# B&R Automation Studio project TD52 (part 58)

#### MFB50Contr_Lib_private.h
```c
/********************************************************************
 * COPYRIGHT -- Bernecker + Rainer Industrie-Elektronik Ges.m.b.H.
 ********************************************************************
 * Program: MFB50Contr_Lib
 * File: MFB50Contr_Lib_private.h
 * Author: 106001702
 * Created: Wed Nov 09 12:46:00 2011
 ********************************************************************
 * Header for program MFB50Contr_Lib
 ********************************************************************
 * Generated with B&R Automation Studio Target for Simulink V4.2
 * (ERT based)
 ********************************************************************/

#ifndef RTW_HEADER_MFB50Contr_Lib_private_h_
#define RTW_HEADER_MFB50Contr_Lib_private_h_
#include "rtwtypes.h"
#include <bur/plctypes.h>
#ifndef __RTWTYPES_H__
#error This file requires rtwtypes.h to be included
#else
#ifdef TMWTYPES_PREVIOUSLY_INCLUDED
#error This file requires rtwtypes.h to be included before tmwtypes.h
#else

/* Check for inclusion of an incorrect version of rtwtypes.h */
#ifndef RTWTYPES_ID_C08S16I32L32N32F1
#error This code was generated with a different "rtwtypes.h" than the file included
#endif                                 /* RTWTYPES_ID_C08S16I32L32N32F1 */
#endif                                 /* TMWTYPES_PREVIOUSLY_INCLUDED */
#endif                                 /* __RTWTYPES_H__ */

#ifndef MIN
#define MIN(a,b)                       ((a) < (b) ? (a) : (b))
#endif

#ifndef MAX
#define MAX(a,b)                       ((a) > (b) ? (a) : (b))
#endif

/* Imported (extern) block parameters */
extern real_T I0AllCyl[21];            /* Variable: I0AllCyl
                                        * Referenced by: '<Root>/inputvariable'
                                        */
extern real_T MFB50ActAllCyl[21];      /* Variable: MFB50ActAllCyl
                                        * Referenced by: '<Root>/inputvariable8'
                                        */
extern real_T MFB50EnPowTh;            /* Variable: MFB50EnPowTh
                                        * Referenced by: '<Root>/Relay'
                                        */
extern real_T MFB50EnSpdTh;            /* Variable: MFB50EnSpdTh
                                        * Referenced by: '<Root>/default 500 (rpm)'
                                        */
extern real_T MFB50GlobRefExt;         /* Variable: MFB50GlobRefExt
                                        * Referenced by: '<Root>/MFB50RefGlobExt (CADafTDC)'
                                        */
extern real_T MFB50RefOffsetAllCyl[21];/* Variable: MFB50RefOffsetAllCyl
                                        * Referenced by: '<Root>/inputvariable20'
                                        */
extern real_T MapIoP2sx[2];            /* Variable: MapIoP2sx
                                        * Referenced by: '<S7>/inputvariable1'
                                        */
extern real_T MapIoP2sy[2];            /* Variable: MapIoP2sy
                                        * Referenced by: '<S7>/inputvariable2'
                                        */
extern real_T MapMFB50oP2sx[2];        /* Variable: MapMFB50oP2sx
                                        * Referenced by: '<S4>/inputvariable1'
                                        */
extern real_T MapMFB50oP2sy[2];        /* Variable: MapMFB50oP2sy
                                        * Referenced by: '<S4>/inputvariable2'
                                        */
extern real_T MapMFB50oT3HPx[2];       /* Variable: MapMFB50oT3HPx
                                        * Referenced by: '<S4>/inputvariable7'
                                        */
extern real_T MapMFB50oT3HPy[2];       /* Variable: MapMFB50oT3HPy
                                        * Referenced by: '<S4>/inputvariable8'
                                        */
extern real_T MapPoP2sx[2];            /* Variable: MapPoP2sx
                                        * Referenced by: '<S7>/inputvariable8'
                                        */
extern real_T MapPoP2sy[2];            /* Variable: MapPoP2sy
                                        * Referenced by: '<S7>/inputvariable9'
                                        */
extern real_T PelAct;                  /* Variable: PelAct
                                        * Referenced by: '<Root>/Pel actual (%)'
                                        */
extern real_T T1_PT1;                  /* Variable: T1_PT1
                                        * Referenced by:
                                        *   '<S9>/timeconst'
                                        *   '<S10>/T1_PT1'
                                        */
extern real_T T3HP_A;                  /* Variable: T3HP_A
                                        * Referenced by: '<Root>/T3HP_A (°C)'
                                        */
extern real_T T3HP_B;                  /* Variable: T3HP_B
                                        * Referenced by: '<Root>/T3HP_B (°C)'
                                        */
extern real_T deadbandNeg;             /* Variable: deadbandNeg
                                        * Referenced by: '<S12>/Constant10'
                                        */
extern real_T deadbandPos;             /* Variable: deadbandPos
                                        * Referenced by: '<S12>/Constant9'
                                        */
extern real_T engSpeed;                /* Variable: engSpeed
                                        * Referenced by: '<Root>/engSpeed (rpm)'
                                        */
extern real_T init_PT1[21];            /* Variable: init_PT1
                                        * Referenced by:
                                        *   '<S9>/Initial value'
                                        *   '<S10>/init_PT1'
                                        */
extern real_T p2s_A;                   /* Variable: p2s_A
                                        * Referenced by: '<Root>/p2s_A (mbar)'
                                        */
extern real_T p2s_B;                   /* Variable: p2s_B
                                        * Referenced by: '<Root>/p2s_B (mbar)'
                                        */
extern real_T uMax;                    /* Variable: uMax
                                        * Referenced by: '<S12>/Constant6'
                                        */
extern real_T uMin;                    /* Variable: uMin
                                        * Referenced by: '<S12>/Constant7'
                                        */
extern int16_T EngOpState;             /* Variable: EngOpState
                                        * Referenced by: '<Root>/inputvariable5'
                                        */
extern boolean_T LoadEnabled;          /* Variable: LoadEnabled
                                        * Referenced by: '<Root>/Load enabled (boolean)'
                                        */
extern boolean_T MFB50ContrEn;         /* Variable: MFB50ContrEn
                                        * Referenced by: '<Root>/inputvariable6'
                                        */
extern boolean_T MFB50MedianEn;        /* Variable: MFB50MedianEn
                                        * Referenced by: '<Root>/MFB50MedianEn'
                                        */
extern boolean_T freezeAllCyl[21];     /* Variable: freezeAllCyl
                                        * Referenced by: '<Root>/inputvariable23'
                                        */
extern boolean_T isFastStart;          /* Variable: isFastStart
                                        * Referenced by: '<Root>/inputvariable4'
                                        */
extern boolean_T isITRetLimpHomeAllCyl[21];/* Variable: isITRetLimpHomeAllCyl
                                            * Referenced by: '<Root>/inputvariable7'
                                            */
extern boolean_T isKnockITRetAllCyl[21];/* Variable: isKnockITRetAllCyl
                                         * Referenced by: '<Root>/inputvariable2'
                                         */
extern boolean_T isSensFailAllCyl[21]; /* Variable: isSensFailAllCyl
                                        * Referenced by: '<Root>/inputvariable3'
                                        */
extern boolean_T isSkipAllCyl[21];     /* Variable: isSkipAllCyl
                                        * Referenced by: '<Root>/inputvariable1'
                                        */
extern boolean_T resetAllCyl[21];      /* Variable: resetAllCyl
                                        * Referenced by: '<Root>/manual reset'
                                        */
extern real_T rt_roundd(real_T u, struct MFB50Contr* inst);

/* Exported functions */
void BINARYSEARCH_real_T(uint32_T *piLeft, uint32_T *piRght, real_T u, const
  real_T *pData, uint32_T iHi, struct MFB50Contr* inst);
void LookUp_real_T_real_T(real_T *pY, const real_T *pYData, real_T u, const
  real_T *pUData, uint32_T iHi, struct MFB50Contr* inst);

#endif                                 /* RTW_HEADER_MFB50Contr_Lib_private_h_ */
```

#### MFB50Contr_Lib_types.h
```c
/********************************************************************
 * COPYRIGHT -- Bernecker + Rainer Industrie-Elektronik Ges.m.b.H.
 ********************************************************************
 * Program: MFB50Contr_Lib
 * File: MFB50Contr_Lib_types.h
 * Author: 106001702
 * Created: Wed Nov 09 12:46:00 2011
 ********************************************************************
 * Header for program MFB50Contr_Lib
 ********************************************************************
 * Generated with B&R Automation Studio Target for Simulink V4.2
 * (ERT based)
 ********************************************************************/

#ifndef RTW_HEADER_MFB50Contr_Lib_types_h_
#define RTW_HEADER_MFB50Contr_Lib_types_h_
#ifndef MIN
#define MIN(a,b)                       ((a) < (b) ? (a) : (b))
#endif

#ifndef MAX
#define MAX(a,b)                       ((a) > (b) ? (a) : (b))
#endif
#endif                                 /* RTW_HEADER_MFB50Contr_Lib_types_h_ */
```

#### rtwtypes.h
```c
/********************************************************************
 * COPYRIGHT -- Bernecker + Rainer Industrie-Elektronik Ges.m.b.H.
 ********************************************************************
 * Program: MFB50Contr_Lib
 * File: rtwtypes.h
 * Author: 106001702
 * Created: Wed Nov 09 12:46:00 2011
 ********************************************************************
 * Header for program MFB50Contr_Lib
 ********************************************************************
 * Generated with B&R Automation Studio Target for Simulink V4.2
 * (ERT based)
 ********************************************************************/

#ifndef __RTWTYPES_H__
#define __RTWTYPES_H__
#ifndef TRUE
# define TRUE                          (1U)
#endif

#ifndef FALSE
# define FALSE                         (0U)
#endif

#ifndef __TMWTYPES__
#define __TMWTYPES__
#include <limits.h>

/*=======================================================================*
 * Target hardware information
 *   Device type: Intel->x86/Pentium
 *   Number of bits:     char:   8    short:   16    long:  32
 *                       long:  32
 *                       native word size:  32
 *   Byte ordering: LittleEndian
 *   Signed integer division rounds to: Zero
 *   Shift right on a signed integer as arithmetic shift: on
 *=======================================================================*/

/*=======================================================================*
 * Fixed width word size data types:                                     *
 *   int8_T, int16_T, int32_T     - signed 8, 16, or 32 bit integers     *
 *   uint8_T, uint16_T, uint32_T  - unsigned 8, 16, or 32 bit integers   *
 *   real32_T, real64_T           - 32 and 64 bit floating point numbers *
 *=======================================================================*/
typedef signed char int8_T;
typedef unsigned char uint8_T;
typedef short int16_T;
typedef unsigned short uint16_T;
typedef long int32_T;
typedef unsigned long uint32_T;
typedef float real32_T;
typedef double real64_T;

/*===========================================================================*
 * Generic type definitions: real_T, time_T, boolean_T, int_T, uint_T,       *
 *                           ulong_T, char_T and byte_T.                     *
 *===========================================================================*/
typedef double real_T;
typedef double time_T;
typedef unsigned char boolean_T;
typedef long int_T;
typedef unsigned long uint_T;
typedef unsigned long ulong_T;
typedef char char_T;
typedef unsigned char uchar_T;
typedef char_T byte_T;

/*=======================================================================*
 * Min and Max:                                                          *
 *   int8_T, int16_T, int32_T     - signed 8, 16, or 32 bit integers     *
 *   uint8_T, uint16_T, uint32_T  - unsigned 8, 16, or 32 bit integers   *
 *=======================================================================*/
#define MAX_int8_T                     ((int8_T)(127))
#define MIN_int8_T                     ((int8_T)(-128))
#define MAX_uint8_T                    ((uint8_T)(255U))
#define MIN_uint8_T                    ((uint8_T)(0U))
#define MAX_int16_T                    ((int16_T)(32767))
#define MIN_int16_T                    ((int16_T)(-32768))
#define MAX_uint16_T                   ((uint16_T)(65535U))
#define MIN_uint16_T                   ((uint16_T)(0U))
#define MAX_int32_T                    ((int32_T)(2147483647))
#define MIN_int32_T                    ((int32_T)(-2147483647-1))
#define MAX_uint32_T                   ((uint32_T)(0xFFFFFFFFU))
#define MIN_uint32_T                   ((uint32_T)(0U))

/* Logical type definitions */
#if (!defined(__cplusplus)) && (!defined(__true_false_are_keywords))
#  ifndef false
#   define false                       (0U)
#  endif

#  ifndef true
#   define true                        (1U)
#  endif
#endif

/*
 * Simulink Coder assumes the code is compiled on a target using a 2's complement representation
 * for signed integer values.
 */
#if ((SCHAR_MIN + 1) != -SCHAR_MAX)
#error "This code must be compiled using a 2's complement representation for signed integer values"
#endif

/* This ID is used to detect inclusion of an incompatible rtwtypes.h */
#define RTWTYPES_ID_C08S16I32L32N32F1
#else                                  /* __TMWTYPES__ */
#define TMWTYPES_PREVIOUSLY_INCLUDED
#endif                                 /* __TMWTYPES__ */

/* Block D-Work pointer type */
typedef void * pointer_T;

/* Simulink specific types */
#ifndef __SIMSTRUC_TYPES_H__
#define __SIMSTRUC_TYPES_H__

/* Trigger directions: falling, either, and rising */
typedef enum {
  FALLING_ZERO_CROSSING = -1,
  ANY_ZERO_CROSSING = 0,
  RISING_ZERO_CROSSING = 1
} ZCDirection;

/* Previous state of a trigger signal */
typedef uint8_T ZCSigState;

/* Initial value of a trigger zero crossing signal */
#define UNINITIALIZED_ZCSIG            0x03U
#define NEG_ZCSIG                      0x02U
#define POS_ZCSIG                      0x01U
#define ZERO_ZCSIG                     0x00U

/* Current state of a trigger signal */
typedef enum {
  FALLING_ZCEVENT = -1,
  NO_ZCEVENT = 0,
  RISING_ZCEVENT = 1
} ZCEventType;

#endif                                 /* __SIMSTRUC_TYPES_H__ */
#endif                                 /* __RTWTYPES_H__ */

#ifndef MIN
#define MIN(a,b)                       ((a) < (b) ? (a) : (b))
#endif

#ifndef MAX
#define MAX(a,b)                       ((a) > (b) ? (a) : (b))
#endif
```

#### MFB50Contr_Lib.c
```c
/********************************************************************
 * COPYRIGHT -- Bernecker + Rainer Industrie-Elektronik Ges.m.b.H.
 ********************************************************************
 * Program: MFB50Contr_Lib
 * File: MFB50Contr_Lib.c
 * Author: 106001702
 * Created: Wed Nov 09 12:46:00 2011
 ********************************************************************
 * Implementation of program MFB50Contr_Lib
 ********************************************************************
 * Generated with B&R Automation Studio Target for Simulink V4.2
 * (ERT based)
 ********************************************************************/
#include "MFB50Contr_Lib.h"
#include "MFB50Contr_Lib_private.h"

/*  Defines */

/*  Data Types */

/**************************** GLOBAL DATA *************************************/
/*  Definitions */

/* Block signals (auto storage) */
struct BlockIO_MFB50Contr_Lib MFB50Contr_Lib_B;

/* Block states (auto storage) */
struct D_Work_MFB50Contr_Lib MFB50Contr_Lib_DWork;

/*  Declarations  */

/***************************** FILE SCOPE DATA ********************************/

/*************************** FUNCTIONS ****************************************/

/* Lookup Binary Search Utility BINARYSEARCH_real_T */
void BINARYSEARCH_real_T(uint32_T *piLeft, uint32_T *piRght, real_T u, const
  real_T *pData, uint32_T iHi, struct MFB50Contr* inst)
{
  /* Find the location of current input value in the data table. */
  *piLeft = 0U;
  *piRght = iHi;
  if (u <= pData[0] ) {
    /* Less than or equal to the smallest point in the table. */
    *piRght = 0U;
  } else if (u >= pData[iHi] ) {
    /* Greater than or equal to the largest point in the table. */
    *piLeft = iHi;
  } else {
    uint32_T i;

    /* Do a binary search. */
    while (( *piRght - *piLeft ) > 1U ) {
      /* Get the average of the left and right indices using to Floor rounding. */
      i = (*piLeft + *piRght) >> 1;

      /* Move either the right index or the left index so that */
      /*  LeftDataPoint <= CurrentValue < RightDataPoint */
      if (u < pData[i] ) {
        *piRght = i;
      } else {
        *piLeft = i;
      }
    }
  }
}

/* Lookup Utility LookUp_real_T_real_T */
void LookUp_real_T_real_T(real_T *pY, const real_T *pYData, real_T u, const
  real_T *pUData, uint32_T iHi, struct MFB50Contr* inst)
{
  uint32_T iLeft;
  uint32_T iRght;
  BINARYSEARCH_real_T( &(iLeft), &(iRght), u, pUData, iHi, inst);

  {
    real_T lambda;
    if (pUData[iRght] > pUData[iLeft] ) {
      real_T num;
      real_T den;
      den = pUData[iRght];
      den = den - pUData[iLeft];
      num = u;
      num = num - pUData[iLeft];
      lambda = num / den;
    } else {
      lambda = 0.0;
    }

    {
      real_T yLeftCast;
      real_T yRghtCast;
      yLeftCast = pYData[iLeft];
      yRghtCast = pYData[iRght];
      yLeftCast += lambda * ( yRghtCast - yLeftCast );
      (*pY) = yLeftCast;
    }
  }
}

real_T rt_roundd(real_T u, struct MFB50Contr* inst)
{
  real_T y;
  if (fabs(u) < 4.503599627370496E+15) {
    if (u >= 0.5) {
      y = floor(u + 0.5);
    } else if (u > -0.5) {
      y = 0.0;
    } else {
      y = ceil(u - 0.5);
    }
  } else {
    y = u;
  }

  return y;
}

/* Model step function */
void MFB50Contr_Lib_step(struct MFB50Contr* inst)
{
  int8_T idx[21];
  int32_T k;
  int8_T idx_0[21];
  int32_T i;
  int32_T j;
  int32_T p;
  int32_T q;
  int32_T qEnd;
  int32_T kEnd;
  real_T rtb_Switch1_e;
  real_T rtb_Switch2;
  boolean_T rtb_Compare;
  real_T rtb_Switch1;
  boolean_T rtb_Switch_k[21];
  int32_T s10_iter;
  int32_T i_0;

  /* Switch: '<S8>/Switch' incorporates:
   *  Constant: '<Root>/inst->engSpeed (rpm)'
   *  Constant: '<S8>/const1'
   */
  if (inst->engSpeed > 0.0) {
    rtb_Switch1 = inst->engSpeed;
  } else {
    rtb_Switch1 = 1.0;
  }

  /* End of Switch: '<S8>/Switch' */

  /* Product: '<S8>/Divide' incorporates:
   *  Constant: '<S8>/const'
   */
  MFB50Contr_Lib_B.Divide = 120.0 / rtb_Switch1;

  /* Switch: '<S8>/Switch2' incorporates:
   *  Constant: '<S8>/const4'
   *  Sum: '<S8>/Add'
   *  Sum: '<S8>/Add1'
   *  UnitDelay: '<S8>/Unit Delay'
   */
  if ((0.01 + MFB50Contr_Lib_DWork.UnitDelay_DSTATE) - MFB50Contr_Lib_B.Divide >=
      0.0) {
    rtb_Switch2 = 0.01;
  } else {
    rtb_Switch2 = 0.01 + MFB50Contr_Lib_DWork.UnitDelay_DSTATE;
  }

  /* End of Switch: '<S8>/Switch2' */

  /* DataTypeConversion: '<S8>/Data Type Conversion' incorporates:
   *  Constant: '<S8>/const4'
   *  Product: '<S8>/Divide2'
   */
  rtb_Switch1 = fmod(rt_roundd(100.0 * rtb_Switch2, inst), 4.294967296E+9);
  MFB50Contr_Lib_B.DataTypeConversion = rtb_Switch1 < 0.0 ? -(int32_T)(uint32_T)
    -rtb_Switch1 : (int32_T)(uint32_T)rtb_Switch1;

  /* Switch: '<Root>/Switch1' incorporates:
   *  Constant: '<Root>/Constant1'
   *  Constant: '<Root>/inputvariable6'
   */
  if (inst->MFB50ContrEn) {
    rtb_Switch1_e = (real_T)MFB50Contr_Lib_B.DataTypeConversion;
  } else {
    rtb_Switch1_e = 99.0;
  }

  /* End of Switch: '<Root>/Switch1' */

  /* MATLAB Function: '<Root>/Median' incorporates:
   *  Constant: '<Root>/inputvariable8'
   */
  /* MATLAB Function 'Median': '<S5>:1' */
  /*  Output */
  /*  y_f: filtered signal - tustin approximation */
  /* '<S5>:1:6' */
  for (s10_iter = 0; s10_iter < 21; s10_iter++) {
    idx[s10_iter] = (int8_T)(s10_iter + 1);
  }

  for (s10_iter = 0; s10_iter <= 18; s10_iter += 2) {
    if (!(inst->MFB50ActAllCyl[s10_iter] <= inst->MFB50ActAllCyl[s10_iter + 1])) {
      idx[s10_iter] = (int8_T)(s10_iter + 2);
      idx[s10_iter + 1] = (int8_T)(s10_iter + 1);
    }
  }

  for (i_0 = 0; i_0 < 21; i_0++) {
    idx_0[i_0] = 1;
  }

  i_0 = 2;
  while (i_0 < 21) {
    i = i_0 << 1;
    j = 1;
    s10_iter = 1 + i_0;
    while (s10_iter < 22) {
      p = j;
      q = s10_iter;
      qEnd = j + i;
      if (qEnd > 22) {
        qEnd = 22;
      }

      k = 0;
      kEnd = qEnd - j;
      while (k + 1 <= kEnd) {
        if (inst->MFB50ActAllCyl[idx[p - 1] - 1] <= inst->MFB50ActAllCyl[idx[q - 1] - 1]) {
          idx_0[k] = idx[p - 1];
          p++;
          if (p == s10_iter) {
            while (q < qEnd) {
              k++;
              idx_0[k] = idx[q - 1];
              q++;
            }
          }
        } else {
          idx_0[k] = idx[q - 1];
          q++;
          if (q == qEnd) {
            while (p < s10_iter) {
              k++;
              idx_0[k] = idx[p - 1];
              p++;
            }
          }
        }

        k++;
      }

      for (s10_iter = 0; s10_iter + 1 <= kEnd; s10_iter++) {
        idx[(j + s10_iter) - 1] = idx_0[s10_iter];
      }

      j = qEnd;
      s10_iter = qEnd + i_0;
    }

    i_0 = i;
  }

  MFB50Contr_Lib_B.y_median = inst->MFB50ActAllCyl[idx[10] - 1];

  /* End of MATLAB Function: '<Root>/Median' */

  /* MATLAB Function: '<Root>/1st order Filter2' incorporates:
   *  Constant: '<S9>/Initial value'
   *  Constant: '<S9>/timeconst'
   *  SignalConversion: '<S1>/TmpSignal ConversionAt SFunction Inport2'
   */
  /* MATLAB Function '1st order Filter2': '<S1>:1' */
  /*  Input */
  /*  y: raw signal */
  /*  parameters */
  /* '<S1>:1:9' */
  /*  time const */
  /* '<S1>:1:10' */
  /*  sample time */
  /* '<S1>:1:11' */
  /*  initial conditions */
  /*  init */
  if (!MFB50Contr_Lib_DWork.y_z_not_empty_p) {
    /* '<S1>:1:14' */
    /* '<S1>:1:15' */
    MFB50Contr_Lib_DWork.y_z_l = inst->init_PT1[0];
    MFB50Contr_Lib_DWork.y_z_not_empty_p = TRUE;

    /* '<S1>:1:16' */
    MFB50Contr_Lib_DWork.y_f_z_i = inst->init_PT1[0];
  }

  /*  Output */
  /*  y_f: filtered signal - tustin approximation */
  /* '<S1>:1:21' */
  MFB50Contr_Lib_B.y_f_e = (((200.0 * inst->T1_PT1 - 1.0) *
    MFB50Contr_Lib_DWork.y_f_z_i + MFB50Contr_Lib_B.y_median) +
    MFB50Contr_Lib_DWork.y_z_l) * (1.0 / (200.0 * inst->T1_PT1 + 1.0));

  /* '<S1>:1:23' */
  MFB50Contr_Lib_DWork.y_z_l = MFB50Contr_Lib_B.y_median;

  /* '<S1>:1:24' */
  MFB50Contr_Lib_DWork.y_f_z_i = MFB50Contr_Lib_B.y_f_e;

  /* End of MATLAB Function: '<Root>/1st order Filter2' */

  /* SwitchCase: '<Root>/Switch Case1' */
  rtb_Switch1 = fmod(rtb_Switch1_e, 4.294967296E+9);
  switch (rtb_Switch1 < 0.0 ? -(int32_T)(uint32_T)-rtb_Switch1 : (int32_T)
          (uint32_T)rtb_Switch1) {
   case 2:
    /* Outputs for IfAction SubSystem: '<Root>/MFB50RefCalc' incorporates:
     *  ActionPort: '<S4>/Action Port'
     */
    /* Dynamic Look-Up Table Block: '<S4>/Lookup Table Dynamic1'
     * Input0  Data Type:  Floating Point real_T
     * Input1  Data Type:  Floating Point real_T
     * Input2  Data Type:  Floating Point real_T
     * Output0 Data Type:  Floating Point real_T
     * Lookup Method: Linear_Endpoint
     *
     */
    LookUp_real_T_real_T( &(MFB50Contr_Lib_B.LookupTableDynamic1_m),
                         inst->MapMFB50oP2sy, MFB50Contr_Lib_B.p2sOut, inst->MapMFB50oP2sx,
                         1U, inst);

    /* S-Function (bur_out): '<S4>/Output1' */
    inst->MFB50RefGlobP2s = MFB50Contr_Lib_B.LookupTableDynamic1_m;

    /* MATLAB Function: '<S4>/T3HPcalc' incorporates:
     *  Constant: '<Root>/inst->T3HP_A (°C)'
     *  Constant: '<Root>/inst->T3HP_B (°C)'
     */
    /* MATLAB Function 'MFB50RefCalc/T3HPcalc': '<S15>:1' */
    /*  Output */
    if (((inst->T3HP_A < 0.0) || (inst->T3HP_A > 1000.0)) && ((inst->T3HP_B < 0.0) || (inst->T3HP_B >
          1000.0))) {
      /* '<S15>:1:5' */
      /* '<S15>:1:6' */
      MFB50Contr_Lib_B.T3HPout = 80.0;
    } else if ((inst->T3HP_A < 0.0) || (inst->T3HP_A > 1000.0)) {
      /* '<S15>:1:7' */
      /* '<S15>:1:8' */
      MFB50Contr_Lib_B.T3HPout = inst->T3HP_B;
    } else if ((inst->T3HP_B < 0.0) || (inst->T3HP_B > 1000.0)) {
      /* '<S15>:1:9' */
      /* '<S15>:1:10' */
      MFB50Contr_Lib_B.T3HPout = inst->T3HP_A;
    } else {
      /* '<S15>:1:12' */
      MFB50Contr_Lib_B.T3HPout = (inst->T3HP_A + inst->T3HP_B) / 2.0;
    }

    /* End of MATLAB Function: '<S4>/T3HPcalc' */

    /* S-Function (bur_out): '<S4>/Output2' */
    inst->T3HPout = MFB50Contr_Lib_B.T3HPout;

    /* Dynamic Look-Up Table Block: '<S4>/Lookup Table Dynamic'
     * Input0  Data Type:  Floating Point real_T
     * Input1  Data Type:  Floating Point real_T
     * Input2  Data Type:  Floating Point real_T
     * Output0 Data Type:  Floating Point real_T
     * Lookup Method: Linear_Endpoint
     *
     */
    LookUp_real_T_real_T( &(MFB50Contr_Lib_B.LookupTableDynamic), inst->MapMFB50oT3HPy,
                         MFB50Contr_Lib_B.T3HPout, inst->MapMFB50oT3HPx, 1U, inst);

    /* S-Function (bur_out): '<S4>/Output6' */
    inst->MFB50RefGlobT3HP = MFB50Contr_Lib_B.LookupTableDynamic;

    /* Switch: '<S4>/Switch1' incorporates:
     *  Constant: '<Root>/inputvariable4'
     *  Constant: '<S4>/Constant1'
     *  Sum: '<S4>/Add2'
     */
    if (inst->isFastStart) {
      rtb_Switch1 = MFB50Contr_Lib_B.LookupTableDynamic +
        MFB50Contr_Lib_B.LookupTableDynamic1_m;
    } else {
      rtb_Switch1 = 0.0;
    }

    /* End of Switch: '<S4>/Switch1' */

    /* MultiPortSwitch: '<S4>/Engine operation state, down .. 0, speed up .. 1, idle (start in load mode) .. 2, load mode .. 3, idle (stop mode) .. 4 island mode .. 5' incorporates:
     *  Constant: '<Root>/inputvariable5'
     *  Constant: '<S4>/IslandCntr'
     *  Constant: '<S4>/MFB50OffsOther'
     *  Constant: '<S4>/MFB50OffsetIsland'
     */
    switch (inst->EngOpState) {
     case 1:
     case 2:
     case 3:
      break;

     case 4:
      rtb_Switch1 = 0.0;
      break;

     case 5:
      rtb_Switch1 = 0.0;
      break;

     default:
      rtb_Switch1 = 0.0;
      break;
    }

    /* End of MultiPortSwitch: '<S4>/Engine operation state, down .. 0, speed up .. 1, idle (start in load mode) .. 2, load mode .. 3, idle (stop mode) .. 4 island mode .. 5' */

    /* Sum: '<S4>/Add1' incorporates:
     *  Constant: '<Root>/MFB50RefGlobExt (CADafTDC)'
     */
    MFB50Contr_Lib_B.Add1 = rtb_Switch1 + inst->MFB50GlobRefExt;

    /* End of Outputs for SubSystem: '<Root>/MFB50RefCalc' */
    break;

   case 1:
    /* Outputs for IfAction SubSystem: '<Root>/PI cntr gain scheduling' incorporates:
     *  ActionPort: '<S7>/Action Port'
     */
    /* MATLAB Function: '<S7>/P2sCalc' incorporates:
     *  Constant: '<Root>/inst->p2s_A (mbar)'
     *  Constant: '<Root>/inst->p2s_B (mbar)'
     */
    /* MATLAB Function 'PI cntr gain scheduling/P2sCalc': '<S16>:1' */
    /*  Inputs (mbar) */
    /*  Output (mbar) */
    if (((inst->p2s_A < 0.0) || (inst->p2s_A > 10000.0)) && ((inst->p2s_B < 0.0) || (inst->p2s_B >
          10000.0))) {
      /* '<S16>:1:6' */
      /* '<S16>:1:7' */
      MFB50Contr_Lib_B.p2sOut = 1000.0;
    } else if ((inst->p2s_A < 0.0) || (inst->p2s_A > 10000.0)) {
      /* '<S16>:1:8' */
      /* '<S16>:1:9' */
      MFB50Contr_Lib_B.p2sOut = inst->p2s_B;
    } else if ((inst->p2s_B < 0.0) || (inst->p2s_B > 10000.0)) {
      /* '<S16>:1:10' */
      /* '<S16>:1:11' */
      MFB50Contr_Lib_B.p2sOut = inst->p2s_A;
    } else {
      /* '<S16>:1:13' */
      MFB50Contr_Lib_B.p2sOut = (inst->p2s_A + inst->p2s_B) / 2.0;
    }

    /* End of MATLAB Function: '<S7>/P2sCalc' */

    /* S-Function (bur_out): '<S7>/Output1' */
    inst->p2sOut = MFB50Contr_Lib_B.p2sOut;

    /* Dynamic Look-Up Table Block: '<S7>/Lookup Table Dynamic1'
     * Input0  Data Type:  Floating Point real_T
     * Input1  Data Type:  Floating Point real_T
     * Input2  Data Type:  Floating Point real_T
     * Output0 Data Type:  Floating Point real_T
     * Lookup Method: Linear_Endpoint
     *
     */
    LookUp_real_T_real_T( &(MFB50Contr_Lib_B.LookupTableDynamic1), inst->MapPoP2sy,
                         MFB50Contr_Lib_B.p2sOut, inst->MapPoP2sx, 1U, inst);

    /* S-Function (bur_out): '<S7>/Output4' */
    inst->P = MFB50Contr_Lib_B.LookupTableDynamic1;

    /* Dynamic Look-Up Table Block: '<S7>/Lookup Table Dynamic2'
     * Input0  Data Type:  Floating Point real_T
     * Input1  Data Type:  Floating Point real_T
     * Input2  Data Type:  Floating Point real_T
     * Output0 Data Type:  Floating Point real_T
     * Lookup Method: Linear_Endpoint
     *
     */
    LookUp_real_T_real_T( &(MFB50Contr_Lib_B.LookupTableDynamic2), inst->MapIoP2sy,
                         MFB50Contr_Lib_B.p2sOut, inst->MapIoP2sx, 1U, inst);

    /* S-Function (bur_out): '<S7>/Output5' */
    inst->I = MFB50Contr_Lib_B.LookupTableDynamic2;

    /* End of Outputs for SubSystem: '<Root>/PI cntr gain scheduling' */
    break;
  }

  /* End of SwitchCase: '<Root>/Switch Case1' */

  /* Relay: '<Root>/Relay' incorporates:
   *  Constant: '<Root>/Pel actual (%)'
   */
  if (inst->PelAct >= inst->MFB50EnPowTh) {
    MFB50Contr_Lib_DWork.Relay_Mode = TRUE;
  } else {
    if (inst->PelAct <= inst->MFB50EnPowTh - 5.0) {
      MFB50Contr_Lib_DWork.Relay_Mode = FALSE;
    }
  }

  /* RelationalOperator: '<S2>/Compare' incorporates:
   *  Constant: '<Root>/default 500 (rpm)'
   *  Constant: '<Root>/inst->engSpeed (rpm)'
   *  Constant: '<S2>/Constant'
   *  Sum: '<Root>/Add'
   */
  rtb_Compare = (inst->engSpeed - inst->MFB50EnSpdTh > 0.0);

  /* Switch: '<Root>/Switch2' incorporates:
   *  Constant: '<Root>/Load enabled (boolean)'
   *  Logic: '<Root>/Logical Operator'
   */
  if ((int32_T)inst->LoadEnabled > 0) {
    /* Relay: '<Root>/Relay' */
    if (MFB50Contr_Lib_DWork.Relay_Mode) {
      i_0 = 1;
    } else {
      i_0 = 0;
    }

    rtb_Compare = ((i_0 != 0) && rtb_Compare);
  }

  /* End of Switch: '<Root>/Switch2' */

  /* Switch: '<Root>/Switch' incorporates:
   *  Constant: '<Root>/manual reset'
   *  Constant: '<Root>/reset all cylinders below speed treshold'
   */
  for (i_0 = 0; i_0 < 21; i_0++) {
    if (rtb_Compare) {
      rtb_Switch_k[i_0] = inst->resetAllCyl[i_0];
    } else {
      rtb_Switch_k[i_0] = TRUE;
    }
  }

  /* End of Switch: '<Root>/Switch' */

  /* SwitchCase: '<Root>/Switch Case' */
  rtb_Switch1 = fmod(rtb_Switch1_e, 4.294967296E+9);
  switch (rtb_Switch1 < 0.0 ? -(int32_T)(uint32_T)-rtb_Switch1 : (int32_T)
          (uint32_T)rtb_Switch1) {
   case 1:
   case 2:
   case 3:
   case 4:
   case 5:
   case 6:
   case 7:
   case 8:
   case 9:
   case 10:
    /* Outputs for IfAction SubSystem: '<Root>/MFB50Controller' incorporates:
     *  ActionPort: '<S3>/Action Port'
     */
    /* Outputs for Iterator SubSystem: '<S3>/MFB50ContrAllCyl' incorporates:
     *  ForIterator: '<S10>/For Iterator'
     */
    for (s10_iter = 0; s10_iter < 2; s10_iter++) {
      /* DataTypeConversion: '<S10>/Data Type Conversion' incorporates:
       *  Constant: '<S10>/Constant1'
       *  Product: '<S10>/Divide'
       *  Sum: '<S10>/Add1'
       */
      rtb_Switch1 = fmod(rt_roundd((real_T)s10_iter * 10.0 + (real_T)
        MFB50Contr_Lib_B.DataTypeConversion, inst), 4.294967296E+9);
      MFB50Contr_Lib_B.DataTypeConversion_o = rtb_Switch1 < 0.0 ? -(int32_T)
        (uint32_T)-rtb_Switch1 : (int32_T)(uint32_T)rtb_Switch1;

      /* Logic: '<S10>/Logical Operator' incorporates:
       *  Constant: '<Root>/inputvariable1'
       *  Constant: '<Root>/inputvariable23'
       *  Constant: '<Root>/inputvariable3'
       *  Constant: '<Root>/inputvariable7'
       *  Selector: '<S10>/Selector2'
       *  Selector: '<S10>/Selector3'
       *  Selector: '<S10>/Selector5'
       *  Selector: '<S10>/Selector7'
       */
      MFB50Contr_Lib_B.LogicalOperator =
        (inst->freezeAllCyl[MFB50Contr_Lib_B.DataTypeConversion_o] ||
         inst->isSkipAllCyl[MFB50Contr_Lib_B.DataTypeConversion_o] ||
         inst->isSensFailAllCyl[MFB50Contr_Lib_B.DataTypeConversion_o] ||
         inst->isITRetLimpHomeAllCyl[MFB50Contr_Lib_B.DataTypeConversion_o]);

      /* S-Function (bur_out): '<S10>/Output1' */
      inst->freezeCyl = MFB50Contr_Lib_B.LogicalOperator;

      /* S-Function (bur_out): '<S10>/Output3' */
      inst->cyl = MFB50Contr_Lib_B.DataTypeConversion_o;

      /* Saturate: '<S10>/Saturation' incorporates:
       *  Constant: '<Root>/inputvariable8'
       *  Selector: '<S10>/Selector'
       */
      if (inst->MFB50ActAllCyl[MFB50Contr_Lib_B.DataTypeConversion_o] >= 50.0) {
        rtb_Switch1_e = 50.0;
      } else if (inst->MFB50ActAllCyl[MFB50Contr_Lib_B.DataTypeConversion_o] <= -50.0)
      {
        rtb_Switch1_e = -50.0;
      } else {
        rtb_Switch1_e = inst->MFB50ActAllCyl[MFB50Contr_Lib_B.DataTypeConversion_o];
      }

      /* End of Saturate: '<S10>/Saturation' */

      /* MATLAB Function: '<S10>/1st order Filter' incorporates:
       *  Constant: '<S10>/inst->T1_PT1'
       *  Constant: '<S10>/Ts'
       *  Constant: '<S10>/inst->init_PT1'
       */
      /* MATLAB Function 'MFB50Controller/MFB50ContrAllCyl/1st order Filter': '<S11>:1' */
      /*  Input */
      /*  y: raw signal */
      /*  parameters */
      /*  T1: time const */
      /*  Ts: sample time */
      /*  init: initial conditions */
      /*  init */
      if (!MFB50Contr_Lib_DWork.y_z_not_empty) {
        /* '<S11>:1:15' */
        /* '<S11>:1:16' */
        MFB50Contr_Lib_DWork.y_z_not_empty = TRUE;

        /* '<S11>:1:17' */
        for (i_0 = 0; i_0 < 21; i_0++) {
          MFB50Contr_Lib_DWork.y_z[i_0] = inst->init_PT1[i_0];
          MFB50Contr_Lib_DWork.y_f_z[i_0] = inst->init_PT1[i_0];
        }
      }

      if (!MFB50Contr_Lib_DWork.y_f_int_not_empty) {
        /* '<S11>:1:19' */
        /* '<S11>:1:20' */
        for (i_0 = 0; i_0 < 21; i_0++) {
          MFB50Contr_Lib_DWork.y_f_int[i_0] = inst->init_PT1[i_0];
        }

        MFB50Contr_Lib_DWork.y_f_int_not_empty = TRUE;
      }

      /*  Output */
      /*  y_f: filtered signal - tustin approximation */
      /* '<S11>:1:25' */
      i_0 = MFB50Contr_Lib_B.DataTypeConversion_o + 1;
      if ((MFB50Contr_Lib_B.DataTypeConversion_o > 0) && (i_0 <= 0)) {
        i_0 = MAX_int32_T;
      }

      i = MFB50Contr_Lib_B.DataTypeConversion_o + 1;
      if ((MFB50Contr_Lib_B.DataTypeConversion_o > 0) && (i <= 0)) {
        i = MAX_int32_T;
      }

      j = MFB50Contr_Lib_B.DataTypeConversion_o + 1;
      if ((MFB50Contr_Lib_B.DataTypeConversion_o > 0) && (j <= 0)) {
        j = MAX_int32_T;
      }

      MFB50Contr_Lib_DWork.y_f_int[i_0 - 1] = (((16.666666666666668 * inst->T1_PT1 -
        1.0) * MFB50Contr_Lib_DWork.y_f_z[i - 1] + rtb_Switch1_e) +
        MFB50Contr_Lib_DWork.y_z[j - 1]) * (1.0 / (16.666666666666668 * inst->T1_PT1 +
        1.0));

      /* '<S11>:1:27' */
      i_0 = MFB50Contr_Lib_B.DataTypeConversion_o + 1;
      if ((MFB50Contr_Lib_B.DataTypeConversion_o > 0) && (i_0 <= 0)) {
        i_0 = MAX_int32_T;
      }

      MFB50Contr_Lib_DWork.y_z[i_0 - 1] = rtb_Switch1_e;

      /* '<S11>:1:28' */
      i_0 = MFB50Contr_Lib_B.DataTypeConversion_o + 1;
      if ((MFB50Contr_Lib_B.DataTypeConversion_o > 0) && (i_0 <= 0)) {
        i_0 = MAX_int32_T;
      }

      i = MFB50Contr_Lib_B.DataTypeConversion_o + 1;
      if ((MFB50Contr_Lib_B.DataTypeConversion_o > 0) && (i <= 0)) {
        i = MAX_int32_T;
      }

      MFB50Contr_Lib_DWork.y_f_z[i_0 - 1] = MFB50Contr_Lib_DWork.y_f_int[i - 1];

      /* '<S11>:1:29' */
      for (i_0 = 0; i_0 < 21; i_0++) {
        MFB50Contr_Lib_B.y_f[i_0] = MFB50Contr_Lib_DWork.y_f_int[i_0];
      }

      /* End of MATLAB Function: '<S10>/1st order Filter' */

      /* Switch: '<S10>/Switch' incorporates:
       *  Constant: '<Root>/inst->MFB50MedianEn'
       */
      if (inst->MFB50MedianEn) {
        rtb_Switch1 = MFB50Contr_Lib_B.y_f_e;
      } else {
        rtb_Switch1 = MFB50Contr_Lib_B.Add1;
      }

      /* End of Switch: '<S10>/Switch' */

      /* Gain: '<S12>/Gain' incorporates:
       *  Constant: '<Root>/inputvariable20'
       *  Selector: '<S10>/Selector4'
       *  Selector: '<S10>/Selector8'
       *  Sum: '<S10>/Sum'
       *  Sum: '<S12>/Sum'
       */
      rtb_Switch1_e = -((rtb_Switch1 +
                         inst->MFB50RefOffsetAllCyl[MFB50Contr_Lib_B.DataTypeConversion_o])
                        - MFB50Contr_Lib_B.y_f[MFB50Contr_Lib_B.DataTypeConversion_o]);

      /* MATLAB Function: '<S12>/PICntr' incorporates:
       *  Constant: '<Root>/inputvariable'
       *  Constant: '<Root>/inputvariable2'
       *  Constant: '<S12>/Constant10'
       *  Constant: '<S12>/Constant6'
       *  Constant: '<S12>/Constant7'
       *  Constant: '<S12>/Constant9'
       *  Constant: '<S12>/Ts1'
       *  Selector: '<S10>/Selector1'
       *  Selector: '<S10>/Selector6'
       */
      /* MATLAB Function 'MFB50Controller/MFB50ContrAllCyl/PI controller/PICntr': '<S13>:1' */
      /*  init */
      if (!MFB50Contr_Lib_DWork.iState_not_empty) {
        /* '<S13>:1:8' */
        /* '<S13>:1:9' */
        for (i_0 = 0; i_0 < 21; i_0++) {
          MFB50Contr_Lib_DWork.iState[i_0] = inst->I0AllCyl[i_0];
        }

        MFB50Contr_Lib_DWork.iState_not_empty = TRUE;
      }

      if (!MFB50Contr_Lib_DWork.uState_not_empty) {
        /* '<S13>:1:14' */
        /* '<S13>:1:15' */
        for (i_0 = 0; i_0 < 21; i_0++) {
          MFB50Contr_Lib_DWork.uState[i_0] = inst->I0AllCyl[i_0];
        }

        MFB50Contr_Lib_DWork.uState_not_empty = TRUE;
      }

      /* '<S13>:1:18' */
      /* '<S13>:1:19' */
      /* '<S13>:1:20' */
      for (i_0 = 0; i_0 < 21; i_0++) {
        MFB50Contr_Lib_B.out[i_0] = MFB50Contr_Lib_DWork.uState[i_0];
        MFB50Contr_Lib_B.ui[i_0] = MFB50Contr_Lib_DWork.iState[i_0];
        MFB50Contr_Lib_B.up[i_0] = MFB50Contr_Lib_DWork.pState[i_0];
      }

      if ((rtb_Switch1_e <= 0.0) &&
          inst->isKnockITRetAllCyl[MFB50Contr_Lib_B.DataTypeConversion_o] &&
          (!MFB50Contr_Lib_B.LogicalOperator)) {
        /* '<S13>:1:22' */
        /* '<S13>:1:23' */
        rtb_Compare = FALSE;
      } else if ((rtb_Switch1_e > 0.0) &&
                 inst->isKnockITRetAllCyl[MFB50Contr_Lib_B.DataTypeConversion_o]) {
        /* '<S13>:1:24' */
        /* '<S13>:1:25' */
        rtb_Compare = TRUE;
      } else {
        /* '<S13>:1:27' */
        rtb_Compare = MFB50Contr_Lib_B.LogicalOperator;
      }

      if ((rtb_Switch1_e >= inst->deadbandNeg) && (rtb_Switch1_e <= inst->deadbandPos)) {
        /* '<S13>:1:31' */
        /* '<S13>:1:32' */
        rtb_Switch1_e = 0.0;
      } else {
        /* '<S13>:1:34' */
      }

      /* '<S13>:1:37' */
      i_0 = MFB50Contr_Lib_B.DataTypeConversion_o + 1;
      if ((MFB50Contr_Lib_B.DataTypeConversion_o > 0) && (i_0 <= 0)) {
        i_0 = MAX_int32_T;
      }

      MFB50Contr_Lib_DWork.pState[i_0 - 1] =
        MFB50Contr_Lib_B.LookupTableDynamic1 * rtb_Switch1_e;

      /* '<S13>:1:38' */
      i_0 = MFB50Contr_Lib_B.DataTypeConversion_o + 1;
      if ((MFB50Contr_Lib_B.DataTypeConversion_o > 0) && (i_0 <= 0)) {
        i_0 = MAX_int32_T;
      }

      i = MFB50Contr_Lib_B.DataTypeConversion_o + 1;
      if ((MFB50Contr_Lib_B.DataTypeConversion_o > 0) && (i <= 0)) {
        i = MAX_int32_T;
      }

      rtb_Switch1 = (0.12 * MFB50Contr_Lib_B.LookupTableDynamic2 * rtb_Switch1_e
                     + MFB50Contr_Lib_DWork.iState[i_0 - 1]) +
        MFB50Contr_Lib_DWork.pState[i - 1];
      if (rtb_Switch_k[MFB50Contr_Lib_B.DataTypeConversion_o]) {
        /* '<S13>:1:40' */
        /* '<S13>:1:41' */
        i_0 = MFB50Contr_Lib_B.DataTypeConversion_o + 1;
        if ((MFB50Contr_Lib_B.DataTypeConversion_o > 0) && (i_0 <= 0)) {
          i_0 = MAX_int32_T;
        }

        i = MFB50Contr_Lib_B.DataTypeConversion_o + 1;
        if ((MFB50Contr_Lib_B.DataTypeConversion_o > 0) && (i <= 0)) {
          i = MAX_int32_T;
        }

        MFB50Contr_Lib_DWork.iState[i_0 - 1] = inst->I0AllCyl[i - 1];

        /* '<S13>:1:42' */
        i_0 = MFB50Contr_Lib_B.DataTypeConversion_o + 1;
        if ((MFB50Contr_Lib_B.DataTypeConversion_o > 0) && (i_0 <= 0)) {
          i_0 = MAX_int32_T;
        }

        i = MFB50Contr_Lib_B.DataTypeConversion_o + 1;
        if ((MFB50Contr_Lib_B.DataTypeConversion_o > 0) && (i <= 0)) {
          i = MAX_int32_T;
        }

        MFB50Contr_Lib_DWork.uState[i_0 - 1] = inst->I0AllCyl[i - 1];

        /* '<S13>:1:43' */
        i_0 = MFB50Contr_Lib_B.DataTypeConversion_o + 1;
        if ((MFB50Contr_Lib_B.DataTypeConversion_o > 0) && (i_0 <= 0)) {
          i_0 = MAX_int32_T;
        }

        MFB50Contr_Lib_DWork.pState[i_0 - 1] = 0.0;
      } else {
        if ((!rtb_Compare) && (rtb_Switch1 > inst->uMin) && (rtb_Switch1 < inst->uMax)) {
          /* '<S13>:1:44' */
          /*  || ((u <= inst->uMin) && (ki * eDead > 0)) || ((u >= inst->uMax) && (ki * eDead < 0))) */
          /* '<S13>:1:45' */
          i_0 = MFB50Contr_Lib_B.DataTypeConversion_o + 1;
          if ((MFB50Contr_Lib_B.DataTypeConversion_o > 0) && (i_0 <= 0)) {
            i_0 = MAX_int32_T;
          }

          i = MFB50Contr_Lib_B.DataTypeConversion_o + 1;
          if ((MFB50Contr_Lib_B.DataTypeConversion_o > 0) && (i <= 0)) {
            i = MAX_int32_T;
          }

          MFB50Contr_Lib_DWork.iState[i_0 - 1] = 0.12 *
            MFB50Contr_Lib_B.LookupTableDynamic2 * rtb_Switch1_e +
            MFB50Contr_Lib_DWork.iState[i - 1];
        }
      }

      /* '<S13>:1:48' */
      i_0 = MFB50Contr_Lib_B.DataTypeConversion_o + 1;
      if ((MFB50Contr_Lib_B.DataTypeConversion_o > 0) && (i_0 <= 0)) {
        i_0 = MAX_int32_T;
      }

      i = MFB50Contr_Lib_B.DataTypeConversion_o + 1;
      if ((MFB50Contr_Lib_B.DataTypeConversion_o > 0) && (i <= 0)) {
        i = MAX_int32_T;
      }

      rtb_Switch1 = MFB50Contr_Lib_DWork.iState[i_0 - 1] +
        MFB50Contr_Lib_DWork.pState[i - 1];
      if (rtb_Switch1 > inst->uMax) {
        /* '<S13>:1:50' */
        /* '<S13>:1:51' */
        rtb_Switch1 = inst->uMax;
      } else {
        if (rtb_Switch1 < inst->uMin) {
          /* '<S13>:1:52' */
          /* '<S13>:1:53' */
          rtb_Switch1 = inst->uMin;
        }
      }

      if (!rtb_Compare) {
        /* '<S13>:1:56' */
        /* '<S13>:1:57' */
        i_0 = MFB50Contr_Lib_B.DataTypeConversion_o + 1;
        if ((MFB50Contr_Lib_B.DataTypeConversion_o > 0) && (i_0 <= 0)) {
          i_0 = MAX_int32_T;
        }

        MFB50Contr_Lib_DWork.uState[i_0 - 1] = rtb_Switch1;
      }

      /* End of MATLAB Function: '<S12>/PICntr' */
    }

    /* End of Outputs for SubSystem: '<S3>/MFB50ContrAllCyl' */
    /* End of Outputs for SubSystem: '<Root>/MFB50Controller' */
    break;
  }

  /* End of SwitchCase: '<Root>/Switch Case' */

  /* S-Function (bur_out): '<Root>/Output' */
  {
    int_T i1;
    const real_T *u0 = MFB50Contr_Lib_B.out;
    for (i1=0; i1 < 21; i1++) {
      inst->ITOffsetAllCyl_u[i1] = u0[i1];
    }
  }

  /* S-Function (bur_out): '<Root>/Output1' */
  {
    int_T i1;
    const real_T *u0 = MFB50Contr_Lib_B.up;
    for (i1=0; i1 < 21; i1++) {
      inst->ITOffsetAllCyl_up[i1] = u0[i1];
    }
  }

  /* S-Function (bur_out): '<Root>/Output2' */
  {
    int_T i1;
    const real_T *u0 = MFB50Contr_Lib_B.ui;
    for (i1=0; i1 < 21; i1++) {
      inst->ITOffsetAllCyl_ui[i1] = u0[i1];
    }
  }

  /* S-Function (bur_out): '<Root>/Output3' */
  inst->clock = MFB50Contr_Lib_B.DataTypeConversion;

  /* S-Function (bur_out): '<Root>/Output6' */
  inst->MFB50RefGlob = MFB50Contr_Lib_B.Add1;

  /* S-Function (bur_out): '<Root>/Output7' */
  {
    int_T i1;
    const real_T *u0 = MFB50Contr_Lib_B.y_f;
    for (i1=0; i1 < 21; i1++) {
      inst->MFB50ActFiltAllCyl[i1] = u0[i1];
    }
  }

  /* S-Function (bur_out): '<Root>/Output8' */
  inst->MFB50MedianFilt = MFB50Contr_Lib_B.y_f_e;

  /* S-Function (bur_out): '<Root>/Output9' */
  inst->MFB50Median = MFB50Contr_Lib_B.y_median;

  /* S-Function (bur_out): '<S8>/Output3' */
  inst->Tcycle = MFB50Contr_Lib_B.Divide;

  /* Update for UnitDelay: '<S8>/Unit Delay' */
  MFB50Contr_Lib_DWork.UnitDelay_DSTATE = rtb_Switch2;
}

/* Model initialize function */
void MFB50Contr_Lib_initialize(struct MFB50Contr* inst)
{
  /* S-Function (bur_out): '<Root>/Output4' */
  inst->ACversion = 1.1;
}

/* Model terminate function */
void MFB50Contr_Lib_terminate(struct MFB50Contr* inst)
{
  /* (no terminate code required) */
}

/*======================== TOOL VERSION INFORMATION ==========================*
 * MATLAB 8.0 (R2012b)20-Jul-2012                                             *
 * Simulink 8.0 (R2012b)20-Jul-2012                                           *
 * Simulink Coder 8.3 (R2012b)20-Jul-2012                                     *
 * Embedded Coder 6.3 (R2012b)20-Jul-2012                                     *
 * Stateflow 8.0 (R2012b)20-Jul-2012                                          *
 * Simulink Fixed Point 7.2 (R2012b)20-Jul-2012                               *
 *============================================================================*/

/*======================= LICENSE IN USE INFORMATION =========================*
 * matlab                                                                     *
 * matlab_coder                                                               *
 * real-time_workshop                                                         *
 * rtw_embedded_coder                                                         *
 * simulink                                                                   *
 *============================================================================*/
```

#### main.c
```c
/********************************************************************
 * COPYRIGHT -- Bernecker + Rainer Industrie-Elektronik Ges.m.b.H.
 ********************************************************************
 * Program: MFB50Contr_Lib
 * File: main.c
 * Author: 106001702
 * Created: Wed Nov 09 12:46:00 2011
 ********************************************************************
 * Implementation of program MFB50Contr_Lib
 ********************************************************************
 * Generated with B&R Automation Studio Target for Simulink V4.2
 * (ERT based)
 ********************************************************************/
#include <bur/plctypes.h>
#include "MFB50Contr_Lib.h"
#include "rtwtypes.h"

/* Defines */
#define SS_TERMINATE 4
#define SS_OUTPUT 3
#define SS_INITIALIZE 2

/*  Data Types */

/**************************** GLOBAL DATA *************************************/
/*  Definitions */

/*  Declarations  */

/***************************** FILE SCOPE DATA ********************************/

/*************************** FUNCTIONS ****************************************/
#ifdef __cplusplus

unsigned long bur_heap_size = 6553500;

#endif

void MFB50Contr(struct MFB50Contr* inst)
{

  switch (inst->ssMethodType)
  {
   case SS_INITIALIZE:
    /* call model initialize function */
    MFB50Contr_Lib_initialize(inst);
    break;

   case SS_OUTPUT:
    /* call model step function */
    MFB50Contr_Lib_step(inst);

    break;

   case SS_TERMINATE:
    /* call model terminate function */
    MFB50Contr_Lib_terminate(inst);
    break;
  }
}

/*****************************************************************************
   Function block sample time: 0.01s
 *****************************************************************************/

/*****************************************************************************
   B&R Automation Studio Target for Simulink Version: A4.4.1 (09-Dec-2014)
 *****************************************************************************/

/*======================== TOOL VERSION INFORMATION ==========================*
 * MATLAB 8.0 (R2012b)20-Jul-2012                                             *
 * Simulink 8.0 (R2012b)20-Jul-2012                                           *
 * Simulink Coder 8.3 (R2012b)20-Jul-2012                                     *
 * Embedded Coder 6.3 (R2012b)20-Jul-2012                                     *
 * Stateflow 8.0 (R2012b)20-Jul-2012                                          *
 * Simulink Fixed Point 7.2 (R2012b)20-Jul-2012                               *
 *============================================================================*/

/*======================= LICENSE IN USE INFORMATION =========================*
 * matlab                                                                     *
 * matlab_coder                                                               *
 * real-time_workshop                                                         *
 * rtw_embedded_coder                                                         *
 * simulink                                                                   *
 *============================================================================*/
```

#### lib_properties.txt
```
For manual assignment to hardware configuration please
add the following additional include directories:

\Logical\MATLAB_includes\R2012b\

And the following additional build options:

-lm -D MODEL=MFB50Contr_Lib -D NUMST=1 -D NCSTATES=0 -D HAVESTDIO -D ONESTEPFCN=1 -D TERMFCN=1 -D MAT_FILE=0 -D MULTI_INSTANCE_CODE=0 -D INTEGER_CODE=0 -D MT=0 -D CLASSIC_INTERFACE=0 -D TID01EQ=0
```

### Library Logical/EngineController/Lib_EC/TEC (IEC) - A new source library

#### TEC.fun - Exported functions and function blocks
```iecst
(********************************************************************
 * COPYRIGHT -- INNIO Company
 ********************************************************************
 * Library: TEC
 * File: TEC.fun
 * Author: CaksM
 * Created: Dezember 09, 2015
 ********************************************************************
 * Functions and function blocks of library TEC
 ********************************************************************)

FUNCTION TIME_TO_SEC : REAL (* Returns the Time value in seconds*)
	VAR_INPUT
		in : TIME;
	END_VAR
END_FUNCTION

FUNCTION Bank_AB : REAL
	VAR_INPUT
		A : REAL;
		B : REAL;
		bA : BOOL;
		bB : BOOL;
	END_VAR
END_FUNCTION

FUNCTION Bank_A : REAL
	VAR_INPUT
		A : REAL;
		B : REAL;
		bA : BOOL;
		bB : BOOL;
	END_VAR
END_FUNCTION

FUNCTION Bank_B : REAL
	VAR_INPUT
		A : REAL;
		B : REAL;
		bA : BOOL;
		bB : BOOL;
	END_VAR
END_FUNCTION
```

#### convert.st
```iecst
(********************************************************************
 * COPYRIGHT -- INNIO Company
 ********************************************************************
 * Package: TEC
 * File: convert.st
 * Author: CaksM
 * Created: Dec 09, 2015
 *******************************************************************)

FUNCTION TIME_TO_SEC

	TIME_TO_SEC := TIME_TO_REAL(in)/1000.0;

END_FUNCTION

FUNCTION Bank_AB
	IF bA AND bB THEN
		Bank_AB		:=	(A + B) / 2.0;
	ELSIF bA THEN
		Bank_AB		:=	A;
	ELSIF bB THEN
		Bank_AB		:=	B;
	ELSE
		Bank_AB		:=	0;
	END_IF
END_FUNCTION

FUNCTION Bank_A
	IF bA THEN
		Bank_A		:=	A;
	ELSIF bB THEN
		Bank_A		:=	B;
	ELSE
		Bank_A		:=	0;
	END_IF
END_FUNCTION

FUNCTION Bank_B
	IF bB THEN
		Bank_B		:=	B;
	ELSIF bA THEN
		Bank_B		:=	A;
	ELSE
		Bank_B		:=	0;
	END_IF
END_FUNCTION
```

### Library Logical/EngineController/Lib_EC/lSS (ANSIC, version 1.00.0)

#### AC_SS_Cust.c
```c
/********************************************************************
 * COPYRIGHT -- Bernecker + Rainer Industrie-Elektronik Ges.m.b.H.
 ********************************************************************
 * Program: AC_SS_Cust
 * File: AC_SS_Cust.c
 * Author: 105055527
 * Created: Thu May 19 13:50:06 2016
 ********************************************************************
 * Implementation of program AC_SS_Cust
 ********************************************************************
 * Generated with B&R Automation Studio Target for Simulink V5.0
 * (ERT based)
 ********************************************************************/
#include "AC_SS_Cust.h"
#include "AC_SS_Cust_private.h"

/*  Defines */

/*  Data Types */

/**************************** GLOBAL DATA *************************************/
/*  Definitions */

/*  Declarations  */

/***************************** FILE SCOPE DATA ********************************/

/*************************** FUNCTIONS ****************************************/

/* Model step function */
void AC_SS_Cust_step(struct BlockIO_AC_SS_Cust *AC_SS_Cust_B, struct D_Work_AC_SS_Cust
                     *AC_SS_Cust_DWork, ExternalOutputs_AC_SS_Cust *AC_SS_Cust_Y, struct SS_Cust* inst)
{
  /* local block i/o variables */
  boolean_T rtb_LogicalOperator2;
  boolean_T rtb_bSS;
  real32_T rtb_DiscreteTimeIntegrator;
  boolean_T rtb_RelationalOperator_e;

  /* S-Function (bur_bus_in): '<Root>/Bus Input' */
  AC_SS_Cust_B->BusInput = inst->in;

  /* Logic: '<S2>/Logical Operator' incorporates:
   *  RelationalOperator: '<S2>/Relational Operator'
   *  RelationalOperator: '<S2>/Relational Operator1'
   *  S-Function (sfix_bitop): '<S2>/Bitwise Operator'
   *  S-Function (sfix_bitop): '<S2>/Bitwise Operator1'
   */
  rtb_bSS = (((AC_SS_Cust_B->BusInput.iSelectAbs & AC_SS_Cust_B->BusInput.iAbs) ==
              AC_SS_Cust_B->BusInput.iSelectAbs) &&
             ((AC_SS_Cust_B->BusInput.iSelectRel & AC_SS_Cust_B->BusInput.iRel) ==
              AC_SS_Cust_B->BusInput.iSelectRel));

  /* Outputs for Atomic SubSystem: '<S2>/TON' */
  /* Logic: '<S3>/Logical Operator2' */
  rtb_LogicalOperator2 = !rtb_bSS;

  /* DiscreteIntegrator: '<S3>/Discrete-Time Integrator' */
  if (rtb_LogicalOperator2 || (AC_SS_Cust_DWork->DiscreteTimeIntegrator_PrevRese
       != 0)) {
    AC_SS_Cust_DWork->DiscreteTimeIntegrator_DSTATE = 0.0F;
  }

  rtb_DiscreteTimeIntegrator = AC_SS_Cust_DWork->DiscreteTimeIntegrator_DSTATE;

  /* RelationalOperator: '<S3>/Relational Operator' incorporates:
   *  DiscreteIntegrator: '<S3>/Discrete-Time Integrator'
   */
  rtb_RelationalOperator_e = (AC_SS_Cust_DWork->DiscreteTimeIntegrator_DSTATE >=
    AC_SS_Cust_B->BusInput.rTi_Del);

  /* Update for DiscreteIntegrator: '<S3>/Discrete-Time Integrator' incorporates:
   *  DataTypeConversion: '<S4>/Conversion'
   *  Logic: '<S3>/Logical Operator'
   *  Logic: '<S3>/Logical Operator1'
   */
  if (!rtb_LogicalOperator2) {
    AC_SS_Cust_DWork->DiscreteTimeIntegrator_DSTATE += (real32_T)
      ((!rtb_RelationalOperator_e) && rtb_bSS) * 0.01F;
  }

  if (rtb_LogicalOperator2) {
    AC_SS_Cust_DWork->DiscreteTimeIntegrator_PrevRese = 1;
  } else {
    AC_SS_Cust_DWork->DiscreteTimeIntegrator_PrevRese = 0;
  }

  /* End of Update for DiscreteIntegrator: '<S3>/Discrete-Time Integrator' */
  /* End of Outputs for SubSystem: '<S2>/TON' */

  /* BusCreator: '<S2>/Bus Creator' incorporates:
   *  Logic: '<S3>/Logical Operator3'
   */
  AC_SS_Cust_Y->out.bSS = rtb_bSS;

  /* Outputs for Atomic SubSystem: '<S2>/TON' */
  AC_SS_Cust_Y->out.bSS_Del = (rtb_RelationalOperator_e && rtb_bSS);

  /* End of Outputs for SubSystem: '<S2>/TON' */
  AC_SS_Cust_Y->out.rET = rtb_DiscreteTimeIntegrator;

  /* S-Function (bur_bus_out): '<Root>/Bus Output' */
  inst->out = AC_SS_Cust_Y->out;
}

/* Model initialize function */
void AC_SS_Cust_initialize(struct SS_Cust* inst)
{
  /* (no initialization code required) */
}

/* Model terminate function */
void AC_SS_Cust_terminate(struct SS_Cust* inst)
{
  /* (no terminate code required) */
}

/*======================== TOOL VERSION INFORMATION ==========================*
 * MATLAB 8.0 (R2012b)20-Jul-2012                                             *
 * Simulink 8.0 (R2012b)20-Jul-2012                                           *
 * Simulink Coder 8.3 (R2012b)20-Jul-2012                                     *
 * Embedded Coder 6.3 (R2012b)20-Jul-2012                                     *
 * Stateflow 8.0 (R2012b)20-Jul-2012                                          *
 *============================================================================*/

/*======================= LICENSE IN USE INFORMATION =========================*
 * matlab                                                                     *
 * matlab_coder                                                               *
 * real-time_workshop                                                         *
 * rtw_embedded_coder                                                         *
 * simulink                                                                   *
 *============================================================================*/
```

#### AC_SS_Cust.h
```c
/********************************************************************
 * COPYRIGHT -- Bernecker + Rainer Industrie-Elektronik Ges.m.b.H.
 ********************************************************************
 * Program: AC_SS_Cust
 * File: AC_SS_Cust.h
 * Author: 105055527
 * Created: Thu May 19 13:50:06 2016
 ********************************************************************
 * Header for program AC_SS_Cust
 ********************************************************************
 * Generated with B&R Automation Studio Target for Simulink V5.0
 * (ERT based)
 ********************************************************************/

#ifndef RTW_HEADER_AC_SS_Cust_h_
#define RTW_HEADER_AC_SS_Cust_h_
#ifndef AC_SS_Cust_COMMON_INCLUDES_
# define AC_SS_Cust_COMMON_INCLUDES_
#include "rtwtypes.h"
#endif                                 /* AC_SS_Cust_COMMON_INCLUDES_ */

#include "AC_SS_Cust_types.h"
#include "lSS.h"

/* Macros for accessing real-time model data structure */
#ifndef rtmGetErrorStatus
# define rtmGetErrorStatus(rtm)        ((rtm)->errorStatus)
#endif

#ifndef rtmSetErrorStatus
# define rtmSetErrorStatus(rtm, val)   ((rtm)->errorStatus = (val))
#endif

#ifndef rtmGetStopRequested
# define rtmGetStopRequested(rtm)      ((void*) 0)
#endif

#ifndef MIN
#define MIN(a,b)                       ((a) < (b) ? (a) : (b))
#endif

#ifndef MAX
#define MAX(a,b)                       ((a) > (b) ? (a) : (b))
#endif

/* Block signals (auto storage) */

/* Block states (auto storage) for system '<Root>' */

/* External outputs (root outports fed by signals with auto storage) */

/* Real-time Model Data Structure */

/* Model entry point functions */
extern void AC_SS_Cust_initialize(struct SS_Cust* inst);
extern void AC_SS_Cust_step(BlockIO_AC_SS_Cust *AC_SS_Cust_B, D_Work_AC_SS_Cust *
  AC_SS_Cust_DWork, ExternalOutputs_AC_SS_Cust *AC_SS_Cust_Y, struct SS_Cust* inst);
extern void AC_SS_Cust_terminate(struct SS_Cust* inst);

/*-
 * The generated code includes comments that allow you to trace directly
 * back to the appropriate location in the model.  The basic format
 * is <system>/block_name, where system is the system number (uniquely
 * assigned by Simulink) and block_name is the name of the block.
 *
 * Use the MATLAB hilite_system command to trace the generated code back
 * to the model.  For example,
 *
 * hilite_system('<S3>')    - opens system 3
 * hilite_system('<S3>/Kp') - opens and selects block Kp which resides in S3
 *
 * Here is the system hierarchy for this model
 *
 * '<Root>' : 'AC_SS_Cust'
 * '<S1>'   : 'AC_SS_Cust/Environment Controller'
 * '<S2>'   : 'AC_SS_Cust/SS_Cust'
 * '<S3>'   : 'AC_SS_Cust/SS_Cust/TON'
 * '<S4>'   : 'AC_SS_Cust/SS_Cust/TON/Data Type Conversion Inherited'
 */
#endif                                 /* RTW_HEADER_AC_SS_Cust_h_ */
```

#### AC_SS_Cust_private.h
```c
/********************************************************************
 * COPYRIGHT -- Bernecker + Rainer Industrie-Elektronik Ges.m.b.H.
 ********************************************************************
 * Program: AC_SS_Cust
 * File: AC_SS_Cust_private.h
 * Author: 105055527
 * Created: Thu May 19 13:50:06 2016
 ********************************************************************
 * Header for program AC_SS_Cust
 ********************************************************************
 * Generated with B&R Automation Studio Target for Simulink V5.0
 * (ERT based)
 ********************************************************************/

#ifndef RTW_HEADER_AC_SS_Cust_private_h_
#define RTW_HEADER_AC_SS_Cust_private_h_
#include "rtwtypes.h"
#include <bur/plctypes.h>
#ifndef __RTWTYPES_H__
#error This file requires rtwtypes.h to be included
#else
#ifdef TMWTYPES_PREVIOUSLY_INCLUDED
#error This file requires rtwtypes.h to be included before tmwtypes.h
#else

/* Check for inclusion of an incorrect version of rtwtypes.h */
#ifndef RTWTYPES_ID_C08S16I32L32N32F1
#error This code was generated with a different "rtwtypes.h" than the file included
#endif                                 /* RTWTYPES_ID_C08S16I32L32N32F1 */
#endif                                 /* TMWTYPES_PREVIOUSLY_INCLUDED */
#endif                                 /* __RTWTYPES_H__ */

#ifndef MIN
#define MIN(a,b)                       ((a) < (b) ? (a) : (b))
#endif

#ifndef MAX
#define MAX(a,b)                       ((a) > (b) ? (a) : (b))
#endif
#endif                                 /* RTW_HEADER_AC_SS_Cust_private_h_ */
```

#### AC_SS_Cust_types.h
```c
/********************************************************************
 * COPYRIGHT -- Bernecker + Rainer Industrie-Elektronik Ges.m.b.H.
 ********************************************************************
 * Program: AC_SS_Cust
 * File: AC_SS_Cust_types.h
 * Author: 105055527
 * Created: Thu May 19 13:50:06 2016
 ********************************************************************
 * Header for program AC_SS_Cust
 ********************************************************************
 * Generated with B&R Automation Studio Target for Simulink V5.0
 * (ERT based)
 ********************************************************************/

#ifndef RTW_HEADER_AC_SS_Cust_types_h_
#define RTW_HEADER_AC_SS_Cust_types_h_
#include "rtwtypes.h"
#ifndef MIN
#define MIN(a,b)                       ((a) < (b) ? (a) : (b))
#endif

#ifndef MAX
#define MAX(a,b)                       ((a) > (b) ? (a) : (b))
#endif

/* Forward declaration for rtModel */
typedef struct tag_RTM_AC_SS_Cust RT_MODEL_AC_SS_Cust;

#endif                                 /* RTW_HEADER_AC_SS_Cust_types_h_ */
```

#### SS_Cust.c
```c
/********************************************************************
 * COPYRIGHT -- Bernecker + Rainer Industrie-Elektronik Ges.m.b.H.
 ********************************************************************
 * Program: AC_SS_Cust
 * File: SS_Cust.c
 * Author: 105055527
 * Created: Thu May 19 13:50:06 2016
 ********************************************************************
 * Implementation of program AC_SS_Cust
 ********************************************************************
 * Generated with B&R Automation Studio Target for Simulink V5.0
 * (ERT based)
 ********************************************************************/
#include <bur/plctypes.h>
#include "AC_SS_Cust.h"
#include "rtwtypes.h"

/* Defines */
#define SS_TERMINATE 4
#define SS_OUTPUT 3
#define SS_INITIALIZE 2

/*  Data Types */

/**************************** GLOBAL DATA *************************************/
/*  Definitions */

/*  Declarations  */

/***************************** FILE SCOPE DATA ********************************/

/*************************** FUNCTIONS ****************************************/
#ifdef __cplusplus

unsigned long bur_heap_size = 6553500;

#endif

void SS_Cust(struct SS_Cust* inst)
{
/*  tag_RTM_AC_SS_Cust* const AC_SS_Cust_M = &(inst)->bur_AC_SS_Cust;*/
	BlockIO_AC_SS_Cust *AC_SS_Cust_B = &(inst)->bur_BlockIO_AC_SS_Cust;
	D_Work_AC_SS_Cust *AC_SS_Cust_DWork = &(inst)->bur_D_Work_AC_SS_Cust;
	ExternalOutputs_AC_SS_Cust *AC_SS_Cust_Y = &(inst)->bur_ExternalOutputs_AC_SS_Cust;

  switch (inst->ssMethodType)
  {
   case SS_INITIALIZE:
    /* call model initialize function */
    AC_SS_Cust_initialize(inst);
    break;

   case SS_OUTPUT:
    /* call model step function */
    AC_SS_Cust_step(AC_SS_Cust_B, AC_SS_Cust_DWork, AC_SS_Cust_Y, inst);

    break;

   case SS_TERMINATE:
    /* call model terminate function */
    AC_SS_Cust_terminate(inst);
    break;
  }
}

/*****************************************************************************
   Function block sample time: 0.01s
 *****************************************************************************/

/*****************************************************************************
   B&R Automation Studio Target for Simulink Version: A5.1.0 (06-May-2016)
 *****************************************************************************/

/*======================== TOOL VERSION INFORMATION ==========================*
 * MATLAB 8.0 (R2012b)20-Jul-2012                                             *
 * Simulink 8.0 (R2012b)20-Jul-2012                                           *
 * Simulink Coder 8.3 (R2012b)20-Jul-2012                                     *
 * Embedded Coder 6.3 (R2012b)20-Jul-2012                                     *
 * Stateflow 8.0 (R2012b)20-Jul-2012                                          *
 *============================================================================*/

/*======================= LICENSE IN USE INFORMATION =========================*
 * matlab                                                                     *
 * matlab_coder                                                               *
 * real-time_workshop                                                         *
 * rtw_embedded_coder                                                         *
 * simulink                                                                   *
 *============================================================================*/
```

#### lSS.fun
```iecst
FUNCTION_BLOCK SS_Cust
	VAR_INPUT
		ssMethodType :  SINT;
		in :  tSS_In_Cust; (**)
	END_VAR
	VAR_OUTPUT
		out :  tSS_Out_Cust; (**)
	END_VAR
	VAR
		bur_BlockIO_AC_SS_Cust :  BlockIO_AC_SS_Cust;
		bur_D_Work_AC_SS_Cust :  D_Work_AC_SS_Cust;
		bur_ExternalOutputs_AC_SS_Cust :  ExternalOutputs_AC_SS_Cust;
		bur_AC_SS_Cust :  tag_RTM_AC_SS_Cust;
	END_VAR
END_FUNCTION_BLOCK

FUNCTION_BLOCK SS
	VAR_INPUT
		ssMethodType :   SINT;
		in :   tSS_In; (**)
	END_VAR
	VAR_OUTPUT
		dbg :   tSS_Out; (**)
		iAbs :   USINT; (*binary data absolute deviation in limits*)
		iRel :   USINT; (*binary data relative deviation in limits*)
	END_VAR
	VAR
		bur_BlockIO_AC_SS :   BlockIO_AC_SS;
		bur_D_Work_AC_SS :   D_Work_AC_SS;
		bur_ExternalOutputs_AC_SS :   ExternalOutputs_AC_SS;
		bur_AC_SS :   tag_RTM_AC_SS;
	END_VAR
END_FUNCTION_BLOCK
```

#### lSS.typ
```iecst
TYPE
	ExternalInputs_AC_SS :  STRUCT
		IN :      tSS_In;
	END_STRUCT;

	ExternalInputs_AC_SS_Cust :  STRUCT
		in :    tSS_In_Cust;
	END_STRUCT;

	tSS_In :  STRUCT
		P2s :    tSS_into; (*Charge pressure*)
		T2s :    tSS_into; (*Charge temperature*)
		T_EG :    tSS_into; (*Exhaust gas temperature*)
		P_Norm :    tSS_into; (*Actual normalized power*)
		Lam :    tSS_into; (*Lambda*)
		N_Norm :    tSS_into; (*Normalized Speed*)
		P_d_Norm :    tSS_into; (*Desired normalized power*)
		IP :    tSS_into; (*Ignition Point*)
		bReset :    BOOL; (*Reset all integrators to zero*)
	END_STRUCT;

	tSS_Out :  STRUCT
		P2s :    tSS_outo; (*Charge pressure*)
		T2s :    tSS_outo; (*Charge temperature*)
		T_EG :    tSS_outo; (*Exhaust gas temperature*)
		P_Norm :    tSS_outo; (*Actual normalized power*)
		Lam :    tSS_outo; (*Lambda*)
		N_Norm :    tSS_outo; (*Normalized speed*)
		P_d_Norm :    tSS_outo; (*Desired normalized power*)
		IP :    tSS_outo; (*Ignition Point*)
	END_STRUCT;

	tSS_into :  STRUCT
		rAct :    REAL; (*actual value*)
		rSet :    REAL; (*target value*)
		rAbsLim :    REAL; (*allowed absolute deviation*)
		rTi_Filt :    REAL; (*Filter time constant for slew rate [s]*)
		rRelLim :    REAL; (*allowed relative deviation*)
	END_STRUCT;

	tSS_outo :  STRUCT
		bAbs :    BOOL; (*actual value is within allowed absolute deviation*)
		bRel :    BOOL; (*actual value is within allowed relative deviation*)
	END_STRUCT;

	rtB_Filter_AC_SS :  STRUCT
		DiscreteTimeIntegrator :   REAL;
	END_STRUCT;

	rtDW_Filter_AC_SS :  STRUCT
		DiscreteTimeIntegrator_DSTATE :   REAL;
		DiscreteTimeIntegrator_PrevRese :   SINT;
	END_STRUCT;

	BlockIO_AC_SS :  STRUCT
		BusInput :   tSS_In;
		Filter_c :   rtB_Filter_AC_SS;
		Filter_n :   rtB_Filter_AC_SS;
		Filter_f :   rtB_Filter_AC_SS;
		Filter :   rtB_Filter_AC_SS;
		Filter_h :   rtB_Filter_AC_SS;
		Filter_e :   rtB_Filter_AC_SS;
		Filter_a :   rtB_Filter_AC_SS;
		Filter_o :   rtB_Filter_AC_SS;
	END_STRUCT;

	D_Work_AC_SS :  STRUCT
		Filter_c :   rtDW_Filter_AC_SS;
		Filter_n :   rtDW_Filter_AC_SS;
		Filter_f :   rtDW_Filter_AC_SS;
		Filter :   rtDW_Filter_AC_SS;
		Filter_h :   rtDW_Filter_AC_SS;
		Filter_e :   rtDW_Filter_AC_SS;
		Filter_a :   rtDW_Filter_AC_SS;
		Filter_o :   rtDW_Filter_AC_SS;
	END_STRUCT;

	rtC_Filter_AC_SS :  STRUCT
		Conversion :   REAL;
	END_STRUCT;

	ConstBlockIO_AC_SS :  STRUCT
		Constant :   REAL;
		Constant_d :   REAL;
		Constant_j :   REAL;
		Constant_h :   REAL;
		Constant_g :   REAL;
		Constant_hq :   REAL;
		Constant_b :   REAL;
		Constant_f :   REAL;
		Filter_c :   rtC_Filter_AC_SS;
		Filter_n :   rtC_Filter_AC_SS;
		Filter_f :   rtC_Filter_AC_SS;
		Filter :   rtC_Filter_AC_SS;
		Filter_h :   rtC_Filter_AC_SS;
		Filter_e :   rtC_Filter_AC_SS;
		Filter_a :   rtC_Filter_AC_SS;
		Filter_o :   rtC_Filter_AC_SS;
	END_STRUCT;

	ConstParam_AC_SS :  STRUCT
		pooled4 :   ARRAY[0..7] OF USINT;
	END_STRUCT;

	ExternalOutputs_AC_SS :  STRUCT
		iAbs :   USINT;
		iRel :   USINT;
		dbg :   tSS_Out;
	END_STRUCT;

	tag_RTM_AC_SS :  STRUCT
		errorStatus :   REFERENCE TO USINT;
	END_STRUCT;

	tSS_In_Cust :  STRUCT
		rTi_Del :   REAL; (*Time interval engine values must be under abs/rel limits to reach steady state*)
		iSelectAbs :   USINT; (*Absolute Steady State for (p2s, T2s, EGT, P_Norm, Lambda, N_Norm, P_d_Norm, IP)*)
		iSelectRel :   USINT; (*Relative Steady State for (p2s, T2s, EGT, P_Norm, Lambda, N_Norm, P_d_Norm, IP)*)
		iAbs :   USINT; (*binary data absolute deviation in limits*)
		iRel :   USINT; (*binary data relative deviation in limits*)
	END_STRUCT;

	tSS_Out_Cust :  STRUCT
		bSS :   BOOL; (*Selected actual and relative values are within allowed limits*)
		bSS_Del :   BOOL; (*Selected actual and relative values are within allowed limits for ime interval rTi_Del*)
		rET :   REAL; (*Elapsed time*)
	END_STRUCT;

	BlockIO_AC_SS_Cust :  STRUCT
		BusInput :  tSS_In_Cust;
	END_STRUCT;

	D_Work_AC_SS_Cust :  STRUCT
		DiscreteTimeIntegrator_DSTATE :  REAL;
		DiscreteTimeIntegrator_PrevRese :  SINT;
	END_STRUCT;

	ExternalOutputs_AC_SS_Cust :  STRUCT
		out :  tSS_Out_Cust;
	END_STRUCT;

	tag_RTM_AC_SS_Cust :  STRUCT
		errorStatus :  REFERENCE TO USINT;
	END_STRUCT;

END_TYPE
```

#### lib_properties.txt
```
For manual assignment to hardware configuration please
add the following additional include directories:

\Logical\MATLAB_includes\R2012b\

And the following additional build options:

-lm -D MODEL=AC_SS_Cust -D NUMST=1 -D NCSTATES=0 -D HAVESTDIO -D ONESTEPFCN=1 -D TERMFCN=1 -D MAT_FILE=0 -D MULTI_INSTANCE_CODE=1 -D INTEGER_CODE=0 -D MT=0 -D CLASSIC_INTERFACE=0 -D TID01EQ=0
```

#### rtwtypes.h
```c
/********************************************************************
 * COPYRIGHT -- Bernecker + Rainer Industrie-Elektronik Ges.m.b.H.
 ********************************************************************
 * Program: AC_SS_Cust
 * File: rtwtypes.h
 * Author: 105055527
 * Created: Thu May 19 13:50:06 2016
 ********************************************************************
 * Header for program AC_SS_Cust
 ********************************************************************
 * Generated with B&R Automation Studio Target for Simulink V5.0
 * (ERT based)
 ********************************************************************/

#ifndef __RTWTYPES_H__
#define __RTWTYPES_H__
#ifndef TRUE
# define TRUE                          (1U)
#endif

#ifndef FALSE
# define FALSE                         (0U)
#endif

#ifndef __TMWTYPES__
#define __TMWTYPES__
#include <limits.h>

/*=======================================================================*
 * Target hardware information
 *   Device type: Intel->x86/Pentium
 *   Number of bits:     char:   8    short:   16    long:  32
 *                       long:  32
 *                       native word size:  32
 *   Byte ordering: LittleEndian
 *   Signed integer division rounds to: Zero
 *   Shift right on a signed integer as arithmetic shift: on
 *=======================================================================*/

/*=======================================================================*
 * Fixed width word size data types:                                     *
 *   int8_T, int16_T, int32_T     - signed 8, 16, or 32 bit integers     *
 *   uint8_T, uint16_T, uint32_T  - unsigned 8, 16, or 32 bit integers   *
 *   real32_T, real64_T           - 32 and 64 bit floating point numbers *
 *=======================================================================*/
typedef signed char int8_T;
typedef unsigned char uint8_T;
typedef short int16_T;
typedef unsigned short uint16_T;
typedef long int32_T;
typedef unsigned long uint32_T;
typedef float real32_T;
typedef double real64_T;

/*===========================================================================*
 * Generic type definitions: real_T, time_T, boolean_T, int_T, uint_T,       *
 *                           ulong_T, char_T and byte_T.                     *
 *===========================================================================*/
typedef double real_T;
typedef double time_T;
typedef unsigned char boolean_T;
typedef long int_T;
typedef unsigned long uint_T;
typedef unsigned long ulong_T;
typedef char char_T;
typedef unsigned char uchar_T;
typedef char_T byte_T;

/*=======================================================================*
 * Min and Max:                                                          *
 *   int8_T, int16_T, int32_T     - signed 8, 16, or 32 bit integers     *
 *   uint8_T, uint16_T, uint32_T  - unsigned 8, 16, or 32 bit integers   *
 *=======================================================================*/
#define MAX_int8_T                     ((int8_T)(127))
#define MIN_int8_T                     ((int8_T)(-128))
#define MAX_uint8_T                    ((uint8_T)(255U))
#define MIN_uint8_T                    ((uint8_T)(0U))
#define MAX_int16_T                    ((int16_T)(32767))
#define MIN_int16_T                    ((int16_T)(-32768))
#define MAX_uint16_T                   ((uint16_T)(65535U))
#define MIN_uint16_T                   ((uint16_T)(0U))
#define MAX_int32_T                    ((int32_T)(2147483647))
#define MIN_int32_T                    ((int32_T)(-2147483647-1))
#define MAX_uint32_T                   ((uint32_T)(0xFFFFFFFFU))
#define MIN_uint32_T                   ((uint32_T)(0U))

/* Logical type definitions */
#if (!defined(__cplusplus)) && (!defined(__true_false_are_keywords))
#  ifndef false
#   define false                       (0U)
#  endif

#  ifndef true
#   define true                        (1U)
#  endif
#endif

/*
 * Simulink Coder assumes the code is compiled on a target using a 2's complement representation
 * for signed integer values.
 */
#if ((SCHAR_MIN + 1) != -SCHAR_MAX)
#error "This code must be compiled using a 2's complement representation for signed integer values"
#endif

/* This ID is used to detect inclusion of an incompatible rtwtypes.h */
#define RTWTYPES_ID_C08S16I32L32N32F1
#else                                  /* __TMWTYPES__ */
#define TMWTYPES_PREVIOUSLY_INCLUDED
#endif                                 /* __TMWTYPES__ */

/* Block D-Work pointer type */
typedef void * pointer_T;

/* Simulink specific types */
#ifndef __SIMSTRUC_TYPES_H__
#define __SIMSTRUC_TYPES_H__

/* Trigger directions: falling, either, and rising */
typedef enum {
  FALLING_ZERO_CROSSING = -1,
  ANY_ZERO_CROSSING = 0,
  RISING_ZERO_CROSSING = 1
} ZCDirection;

/* Previous state of a trigger signal */
typedef uint8_T ZCSigState;

/* Initial value of a trigger zero crossing signal */
#define UNINITIALIZED_ZCSIG            0x03U
#define NEG_ZCSIG                      0x02U
#define POS_ZCSIG                      0x01U
#define ZERO_ZCSIG                     0x00U

/* Current state of a trigger signal */
typedef enum {
  FALLING_ZCEVENT = -1,
  NO_ZCEVENT = 0,
  RISING_ZCEVENT = 1
} ZCEventType;

#endif                                 /* __SIMSTRUC_TYPES_H__ */
#endif                                 /* __RTWTYPES_H__ */

#ifndef MIN
#define MIN(a,b)                       ((a) < (b) ? (a) : (b))
#endif

#ifndef MAX
#define MAX(a,b)                       ((a) > (b) ? (a) : (b))
#endif
```
